TYPE PLC_TO_UI :
STRUCT
	X_MCSPos : REAL;
	Y_MCSPos : REAL;
	Z_MCSPos : REAL;
	M1_ACSPos : REAL;
	M2_ACSPos : REAL;
	M3_ACSPos : REAL;
	AllAxisEnabled : BOOL;
	AxisError : BOOL;
	KinematicGroupError : BOOL;	
	KinematicGroupingReady : BOOL;
	NCIAxisGrouped : BOOL;
	NCIAXisError : BOOL;
	NCIInterpreterState : UDINT;
	PartProgramLine1 : STRING(80);
	PartProgramLine2 : STRING(80);
	PartProgramLine3 : STRING(80);
END_STRUCT
END_TYPE

(* stored: Version 1.1.0.1, ProductVersion 3.1.4024.12
   DUT PLC_TO_UI: Id {f9012504-93dc-4be8-a8ba-76d0ce4261c0} *)
